# B&R Automation Studio project AxisBasic
Automation Studio 

## Configuration ARM

### Task classes (Cpu.sw)
```
Cyclic#1 (cycle 10000 us, tolerance 10000 us):
  FirstInitP <- Infrastructure.FirstInitProg.prg
Cyclic#3 (cycle 50000 us, tolerance 50000 us):
  AxisBasic <- MotionControl.AxisBasic.prg
Cyclic#4 (cycle 100000 us, tolerance 100000 us):
  MachinePro <- MachineControl.MachineProg.prg
Cyclic#8 (cycle 10000 us, tolerance 30000000 us):
  ErrorProg <- Diagnostics.ErrorProg.prg
  MachineHMI <- MachineControl.MachineHMI.prg
DataObjects: Acp10sys
Binaries: udbdef, FWRules, TCData, acp10cfg, Acp10map, iomap, asfw, Role, sysconf, arconfig, ashwd, User, ashwac
Libraries: operator, runtime, astime, AsIecCon, sys_lib, AsBrStr, ArEventLog, AsBrWStr, Acp10_MC, Acp10man, Acp10par, NcGlobal, brsystem, standard, FileIO, AsArLog, asstring, AxisLib, persist, csvfilelib, fiowrap, stringext, hmitools, ringbuflib, logthat, piper, errorlib, vartools, axiserrlib, powerlnk
```

### Hardware
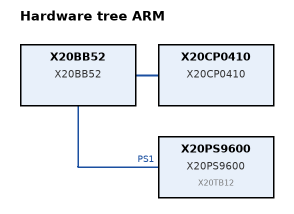
```
X20BB52 : X20BB52 v1.2.0.0
X20CP0410 : X20CP0410 v1.5.0.0  [SL -> X20BB52.SL1]
  Connector IF2:
    ActivateDevice = 1
  ConfigurationID = ServoMgr_ARM
  PermanentPvSize = 1000
  RemanentGlobalPvSize = 5000
  VolatileGlobalPvSize = 300000
  TimerDeviceType = SWIOTIMER
  Cyclic1Duration = 10000
  Cyclic1Tolerance = 10000
  Cyclic2Duration = 20000
  Cyclic2Tolerance = 20000
  Cyclic3Duration = 50000
  Cyclic3Tolerance = 50000
  Cyclic4Duration = 100000
  Cyclic4Tolerance = 100000
  Cyclic5Duration = 200000
  Cyclic5Tolerance = 200000
  Cyclic6Duration = 500000
  Cyclic6Tolerance = 500000
  Cyclic7Duration = 1000000
  Cyclic7Tolerance = 1000000
  Cyclic8Duration = 10000
  Cyclic8Tolerance = 30000000
  FileDevice1
  FileDeviceName1 = USER
  FileDevicePath1 = USER_PATH
X20PS9600 : X20PS9600 v1.6.0.0  [PS -> X20BB52.PS1; SS1 -> X20TB12.SS]
X20TB12 : X20TB12 v1.0.0.0
```

## Configuration Intel

### Task classes (Cpu.sw)
```
Cyclic#1:
  FirstInitP <- Infrastructure.FirstInitProg.prg
Cyclic#3:
  AxisBasic <- MotionControl.AxisBasic.prg
Cyclic#4:
  MachinePro <- MachineControl.MachineProg.prg
Cyclic#8:
  ErrorProg <- Diagnostics.ErrorProg.prg
  MachineHMI <- MachineControl.MachineHMI.prg
DataObjects: Acp10sys
Binaries: udbdef, FWRules, TCData, acp10cfg, Acp10map, iomap, asfw, Role, sysconf, arconfig, ashwd, User, ashwac
Libraries: operator, sys_lib, AsBrStr, runtime, ArEventLog, astime, AsBrWStr, brsystem, Acp10man, Acp10par, NcGlobal, standard, FileIO, AsArLog, AxisLib, asstring, Acp10_MC, piper, persist, csvfilelib, fiowrap, vartools, errorlib, hmitools, ringbuflib, logthat, stringext, axiserrlib, powerlnk, asieccon
```

## Logical view

Binary libraries used (declarations not repeated): Acp10par 5.17.1, AxisLib, persist, csvfilelib, fiowrap, piper 0.01.8, vartools 0.11.4, AxisErrLib, errorlib, hmitools, ringbuflib, stringext, logthat, NcGlobal 5.17.1

### Infrastructure.var
```iecst
(*Constants for number of persisters and permanent memory chunks*)
VAR CONSTANT
	NUM_PERSISTERS : USINT := 4;
	MAI_PERSISTERS : USINT := NUM_PERSISTERS-1;
END_VAR
(*Persisters to handle memory management*)
VAR
	gSimulation: BOOL;
	gPersister : ARRAY[0..MAI_PERSISTERS] OF Persistence_typ;
	gPermBackup : ARRAY[0..MAI_PERSISTERS] OF CSVFileMgr_typ;
END_VAR
VAR RETAIN
	gDataValid : ARRAY[0..MAI_PERSISTERS] OF BOOL;
END_VAR
(*Permanent memory chunks*)
VAR RETAIN
	gPermHomeData : ARRAY[0..999] OF USINT;
	gPermAxisPars : ARRAY[0..999] OF USINT;
	gPermAxisCfgs : ARRAY[0..999] OF USINT;
	gPermConfiguration : ARRAY[0..999] OF USINT;
END_VAR
```

- Acp10err-en.txt (not shown)

### MachineControl.var
```iecst
(********************************************************************
 * COPYRIGHT -- Automation Resources Group
 ********************************************************************
 * Package: MachineControl
 * File: MachineControl.var
 * Author: David Blackburn
 * Created: November 10, 2011
 ********************************************************************
 * Variables of package MachineControl
 ********************************************************************)
VAR
	gMachine : Piper_typ := (0);
END_VAR
VAR RETAIN
	BootTime : TIME;
END_VAR
VAR
	gActiveMode : MODE_MACHINE_ENUM := MODE_MACHINE_AUTO;
	gRequestedMode : MODE_MACHINE_ENUM := MODE_MACHINE_AUTO;
END_VAR
```

### Program Logical/MachineControl/cPiperModuleTemplate

#### Cyclic.c
```c
/********************************************************************
 * COPYRIGHT --
 ********************************************************************
 * Program: cPiperModuleTemplate
 * File: cPiperModuleTemplateCyclic.c
 * Author: dfblackburn
 * Created: April 06, 2016
 ********************************************************************
 * Implementation of program cPiperModuleTemplate
 ********************************************************************/

#include <bur/plctypes.h>

#ifdef _DEFAULT_INCLUDES
	#include <AsDefault.h>
#endif

// Function prototype for piper interface
void PiperModuleInterface();

void _CYCLIC ProgramCyclic(void)
{

	// Call PiperModuleInterface to interface with the rest of the machine
	PiperModuleInterface();

	//Put your code here

}
```

#### PiperInterface.c
```c
/********************************************************************
 * COPYRIGHT --
 ********************************************************************
 * Program: ServoProg
 * File: PiperModuleInterface.c
 * Author: dfblackburn
 * Created: April 01, 2016
 *******************************************************************/

#include <bur/plctypes.h>
#ifdef _DEFAULT_INCLUDES
#include <AsDefault.h>
#endif

#include <string.h>

void PiperModuleInterface() {

	// Give this module a name so it is easier to debug
	strcpy(ModuleInterface.ModuleName, "Name");

	// Add a module to the Piper
	Module.ModuleInterface = &ModuleInterface;
	Module.Piper = &gMachine;
	Piper_Module_Fub(&Module);

	// Handle any machine states that this module needs to respond to
	switch (ModuleInterface.PiperState) {

		//case MACH_ST_BOOTING:
		//case MACH_ST_STOPPED:
		//case MACH_ST_RESETTING:
		//case MACH_ST_IDLE:
		//case MACH_ST_STARTING:
		//case MACH_ST_EXECUTE:
		//case MACH_ST_COMPLETING:
		//case MACH_ST_COMPLETE:
		//case MACH_ST_HOLDING:
		//case MACH_ST_HELD:
		//case MACH_ST_UNHOLDING:
		//case MACH_ST_SUSPENDING:
		//case MACH_ST_SUSPENDED:
		//case MACH_ST_UNSUSPENDING:
		//case MACH_ST_STOPPING:
		//case MACH_ST_ABORTING:
		//case MACH_ST_ABORTED:
		//case MACH_ST_CLEARING:

		case MACH_ST_BYPASSED: break;

		default: ModuleInterface.ModuleResponse = ModuleInterface.PiperState;

	} // switch(PiperState)

} // PiperModuleInterface()
```

### MachineProg.var
```iecst
(********************************************************************
 * COPYRIGHT -- Automation Resources Group
 ********************************************************************
 * Program: MachineProg
 * File: MachineProg.var
 * Author: David Blackburn
 * Created: November 10, 2011
 ********************************************************************
 * Local variables of program MachineProg
 ********************************************************************)
VAR
	HMIMachineCMD : Machine_HMI_CMD_typ := (0);
	HMIMachineState : Machine_HMI_State_typ := (0);
END_VAR
```

- Program Logical/MachineControl/PiperModuleTemplate (IEC) (no source held here)

Listed in the project but not available here: Logical/MachineControl/PiperModuleTemplate/Cyclic.st, Logical/MachineControl/PiperModuleTemplate/PiperModule.var, Logical/MachineControl/PiperModuleTemplate/PiperInterface.st
